TYPE ST_Actor :
    STRUCT
		(* EL2004 - Diguital Out*)
        operatingStateCompressor 	AT %Q* : BOOL;  (* Status des Verdichters: Ein/Aus *)
        operatingStateWaterPump 	AT %Q* : BOOL;  (* Status der Heizungspumpe: Ein/Aus *)
    END_STRUCT
END_TYPE

(* stored: Version 1.1.0.1
   DUT ST_Actor: Id {4250c58b-cb45-4ad1-becf-6a39481befe9} *)
